// TwinCAT 3 PLC project TransportA
// ProgramVersion: 3.1.4023.0
// libraries:
//   Tc2_MC2, * (Beckhoff Automation GmbH)
//   Tc2_Standard, * (Beckhoff Automation GmbH)
//   Tc2_System, * (Beckhoff Automation GmbH)
//   Tc3_Module, * (Beckhoff Automation GmbH)
// project tree:
//   / PlcTask.TcTTO
//   POUs/ MAIN.TcPOU, TransportSystem.TcPOU
// (motion and I/O tree: see PLC project bohrmachine)
// real-time tasks:
//   TASK PlcTask: cycle T#10ms, priority 20, ADS port 350
//   TASK PlcTask1: cycle T#10ms, priority 21, ADS port 351
//   TASK PlcTask2: cycle T#10ms, priority 22, ADS port 352
//   TASK PlcTask3: cycle T#10ms, priority 23, ADS port 353
//   TASK ControllerTask: cycle T#10ms, priority 1, ADS port 354
// variable links:
//   TransportA/TransportA Instance <-> NC-Task 1 SAF/Axes/TransportA
//     PlcTask Inputs/MAIN.fbTransport.axisTransportA.NcToPlc <-> Outputs/ToPlc
//     PlcTask Outputs/MAIN.fbTransport.axisTransportA.PlcToNc <-> Inputs/FromPlc
//   TransportA/TransportA Instance <-> TransportB/TransportB Instance
//     PlcTask Outputs/MAIN.fbTransport.rActVelocity <-> PlcTask Inputs/MAIN.fbTransportSlave.rMasterVelocity
//   TransportA/TransportA Instance <-> Controller/Controller_Obj1 (ModuleController)
//     PlcTask Outputs/MAIN.fbTransport.eZustand <-> TransportA/State
//     PlcTask Outputs/MAIN.fbTransport.objID <-> InputIPointers/oidTransportA

CONFIGURATION TransportA
    RESOURCE PLC ON TwinCAT3
        TASK PlcTask(INTERVAL := T#10ms, PRIORITY := 21);
        PROGRAM MAIN WITH PlcTask : MAIN;
    END_RESOURCE
END_CONFIGURATION

// ---- POUs/MAIN.TcPOU
PROGRAM MAIN
VAR
	fbTransport: TransportSystem('MAIN.TPS_A');
END_VAR

fbTransport();

END_PROGRAM

// ---- POUs/TransportSystem.TcPOU
{attribute 'c++_compatible'}
FUNCTION_BLOCK TransportSystem EXTENDS TcBaseModuleRegistered IMPLEMENTS I_Transport
VAR_INPUT
END_VAR
VAR_OUTPUT
END_VAR
VAR
	// ===== Motion Control =====
	fbMc_MoveVelocity: MC_MoveVelocity;	// continous motion
	fbMc_Stop: MC_Stop;					// stop
	fbMc_Power: MC_Power;				// power
	axisTransportA: AXIS_REF;			// Master axis
	
	// ==== States ====
	eZustand AT %Q*: E_STATES_TRANSPORT_A := E_STATES_TRANSPORT_A.Stopped;	// aktueller Zustand
	bReady: BOOL := FALSE;				// Achse bereit?
	rVelocity: LREAL := 100;			// Velocity (default: 100mm/s)

	// ==== Outputs ====
	rActVelocity AT %Q*: LREAL;				// Actual Velocity output
END_VAR

// ==== Inputs ====
axisTransportA.ReadStatus();

// ==== Outputs ====
// aktuelle Geschwindigkeit
rActVelocity := axisTransportA.NcToPlc.ActVelo;

// ==== Statemachine ====
CASE eZustand OF
	E_STATES_TRANSPORT_A.Starting:
		THIS^.Starting();

	E_STATES_TRANSPORT_A.Started:
		// idle
	
	E_STATES_TRANSPORT_A.Stopping:
		THIS^.Stopping();
	
	E_STATES_TRANSPORT_A.Stopped:
		// idle
	
END_CASE

METHOD FB_reinit : BOOL
VAR_INPUT
END_VAR
SUPER^.FB_reinit();
END_METHOD

{attribute 'TcTypeSystem'}
{attribute 'no-analysis'}
{attribute 'c++_compatible'}
{attribute 'minimal_input_size' := '4'}
{attribute 'pack_mode' := '4'}
METHOD Start : HRESULT
VAR_INPUT
	rVelocity : LREAL;
END_VAR
CASE eZustand OF
	E_STATES_TRANSPORT_A.STARTING:
		Start := S_PENDING;
		
	E_STATES_TRANSPORT_A.STARTED:
		Start := S_OK;
	
	ELSE
		THIS^.rVelocity := rVelocity;
		eZustand := E_STATES_TRANSPORT_A.Starting;
		Start := S_PENDING;
END_CASE
END_METHOD

METHOD Starting : BOOL
VAR_INPUT
END_VAR
// Achse starten und wenn Sie bereit ist, auf gegebene Geschwindigkeit ziehen
// MC_POWER -> MC_MoveVelocity

// TODO jeden Baustein auf Fehler prüfen, evtl allgemeinen Zustand Error einführen

// Achse ist nicht bereit (nicht mit MC_Power gestartet)
IF NOT fbMc_Power.Status THEN
	fbMc_Power(
		Axis := axisTransportA,
		Enable := TRUE,
		Enable_Positive := TRUE
	);
ELSE // Achse ist bereit und beschleunigt auf Zielgeschwindigkeit
	fbMc_MoveVelocity(
		Execute := TRUE,
		Axis := axisTransportA,
		Direction := MC_Direction.MC_Positive_Direction,
		Velocity := rVelocity
	);

	// Achse hat Zielgeschwindigkeit erreicht => Zustand: Started
	IF fbMc_MoveVelocity.InVelocity THEN
		THIS^.eZustand := E_STATES_TRANSPORT_A.Started;
	END_IF	
END_IF


// TODO IF fbMc_Power.Error THEN ... log Error Event + Zustand: Error
END_METHOD

{attribute 'TcTypeSystem'}
{attribute 'no-analysis'}
{attribute 'c++_compatible'}
{attribute 'minimal_input_size' := '4'}
{attribute 'pack_mode' := '4'}
METHOD Stop : HRESULT
CASE eZustand OF
	E_STATES_TRANSPORT_A.STOPPED:
		Stop := S_OK;
		
	E_STATES_TRANSPORT_A.STOPPING:
		Stop := S_PENDING;
		
	ELSE
		eZustand := E_STATES_TRANSPORT_A.Stopping;
		Stop := S_PENDING;
		
END_CASE
END_METHOD

METHOD PRIVATE Stopping : BOOL
VAR_INPUT
END_VAR
//VAR_INST
//	bAxisIsStopped: BOOL := FALSE;
//END_VAR
IF NOT axisTransportA.Status.StandStill THEN
//IF NOT bAxisIsStopped THEN
	// Achse wird gestoppt
	fbMc_Stop(
		Axis := axisTransportA,
		Execute := TRUE
	);
	
	// Achse wurde gestoppt
	IF fbMc_Stop.Done THEN
//		bAxisIsStopped := TRUE;
		// MC_Stop.Done = TRUE && MC_Stop(Execute := FALSE) => Standstill
		fbMc_Stop(
			Axis := axisTransportA,
			Execute := FALSE
		);
	END_IF
ELSE
	// Nach Stop (Standstill), Achse wieder durch Execute := FALSE entriegeln
	fbMc_Stop(
		Axis := axisTransportA,
		Execute := FALSE
	);
	IF NOT fbMc_Stop.Busy THEN
		// Achse wurde wieder entriegelt
		
		// einmal falsen
		fbMc_MoveVelocity(
			Axis := axisTransportA,
			Execute := FALSE
		);
//		bAxisIsStopped := FALSE;
		eZustand := E_STATES_TRANSPORT_A.Stopped;
	END_IF
END_IF
END_METHOD

{attribute 'TcTypeSystem'}
{attribute 'no-analysis'}
{attribute 'c++_compatible'}
{attribute 'minimal_input_size' := '4'}
{attribute 'pack_mode' := '4'}
METHOD TcQueryInterface : HRESULT
VAR_INPUT
	iid	: REFERENCE TO IID;
	pipItf	: POINTER TO PVOID;
END_VAR
VAR
	ipTPS: I_Transport;
END_VAR
IF GuidsEqual(ADR(iid), ADR(TC_GLOBAL_IID_LIST.IID_I_Transport)) THEN
	ipTPS := THIS^;
	pipItf^ := ITCUNKNOWN_TO_PVOID(ipTPS);
	TcAddRef();
	TcQueryInterface := S_OK;
ELSE
	TcQueryInterface := SUPER^.TcQueryInterface(iid, pipItf);
END_IF
END_METHOD

END_FUNCTION_BLOCK
